//Axis FB template, inherited Execute, Busy etc from FbBase   
FUNCTION_BLOCK AxFbBase EXTENDS FbBase 
VAR_INPUT
	rAxis													: REFERENCE TO AXIS_REF := 0; //Reference to AXIS_REF 
END_VAR
VAR_IN_OUT
END_VAR
VAR_OUTPUT
	Active													: BOOL ; // If the axis movement is controlled by several functions, the Active output of each block indicates that the axis executes the command. 
	CmdAborted												: BOOL ; // TRUE if a command is interrupted through another block (Busy and Error = FALSE)
	ErrorText												: STRING(40); //Error text with name of internal used FB which causes the error
END_VAR
VAR 
	LastErrorId												: UDINT := 0; //Last error id
END_VAR

END_FUNCTION_BLOCK

(* stored: Version 1.1.0.1, ProductVersion 3.1.4024.3
   POU AxFbBase: Id {d5ae11fd-111e-4a31-8bab-919faba6d9fa}, SpecialFunc None *)
